{attribute wpf [Container(Layout.GroupBox)]}
TYPE GroupBox_other_other :
STRUCT
	{attribute addProperty Name "<#Stack#>"}
	_stack_other: Stack_other;
	{attribute addProperty Name "<#UniformGrid#>"}
	_uniformGrid_other: UniformGrid_other;
	{attribute addProperty Name "<#Wrap#>"}
	_wrap_other: Wrap_other;
	{attribute addProperty Name "<#Tabs#>"}
	_tabs_other: Tabs_other;
	{attribute addProperty Name "<#Border#>"}
	_border_other: Border_other;
	{attribute addProperty Name "<#GroupBox#>"}
	_groupBox_other: GroupBox_other;
	{attribute addProperty Name "<#Scroll#>"}
	_scroll_other: Scroll_other;
END_STRUCT
END_TYPE

(* stored: Version 1.1.0.1, ProductVersion 3.1.4024.9
   DUT GroupBox_other_other: Id {e36516ac-ef7c-4a38-ad82-264f9556ac31} *)
